FUNCTION_BLOCK PUBLIC FB_Vector3 EXTENDS ExternalStaticMatrix
VAR_INPUT
END_VAR
VAR_OUTPUT
END_VAR
VAR
	data_array : ARRAY [0..2] OF LREAL;
END_VAR

METHOD FB_init : BOOL
VAR_INPUT
	bInitRetains : BOOL; // if TRUE, the retain variables are initialized (warm start / cold start)
	bInCopyCode : BOOL;  // if TRUE, the instance afterwards gets moved into the copy code (online change)
END_VAR
VAR
END_VAR
Init(ADR(data_array), 3, 1);
Clear();
END_METHOD

PROPERTY PUBLIC X : LREAL
GET
X := GetI(0);
END_GET
SET
SetI(0, X);
END_SET
END_PROPERTY

PROPERTY PUBLIC Y : LREAL
GET
Y := GetI(1);
END_GET
SET
SetI(1, Y);
END_SET
END_PROPERTY

PROPERTY PUBLIC Z : LREAL
GET
Z := GetI(2);
END_GET
SET
SetI(2, Z);
END_SET
END_PROPERTY

END_FUNCTION_BLOCK

(* stored: Version 1.1.0.1, ProductVersion 3.1.4024.9
   POU FB_Vector3: Id {451d287b-3f5c-4ee8-81d1-8c7b4ee0b84c}, SpecialFunc None
   Method FB_init: Id {98e9d8da-9aa5-408d-bb08-73efd9a04a3e}
   Property X: Id {148ce7f6-8faf-47c9-a468-0eed359e82ce}
   Get Get: Id {8cba302a-763f-48ad-bb0c-36801daf1f68}
   Set Set: Id {2c9693eb-4139-4ea9-a8ec-a834c5e634dd}
   Property Y: Id {87c9e8a4-dd3b-4c10-93f8-e58f46effca9}
   Get Get: Id {4b160276-4b07-4657-903f-7c1e45a9a03b}
   Set Set: Id {13f78087-e5c4-4679-a23a-c48d92ac0da9}
   Property Z: Id {18afd8ba-4aa8-4180-bc7b-cda30301f6b1}
   Get Get: Id {9af28f71-6afa-4482-af94-3a7c7276df86}
   Set Set: Id {6dd386f6-8894-4825-b5c6-cad0d7bf6850} *)
